FUNCTION Grey_To_Bin : INT // convert 4 bit grey code into 8 bit binary code
VAR_INPUT
	GreyBit0 : BOOL := FALSE ;
	GreyBit1 : BOOL := FALSE ;
	GreyBit2 : BOOL := FALSE ;
	GreyBit3 : BOOL := FALSE ;
END_VAR
VAR
	TempInt : INT ; // temporary 
END_VAR

// convert grey code into binary
TempInt.3 	:= GreyBit3 ;
TempInt.2	:= GreyBit3 	XOR GreyBit2 ;
TempInt.1	:= TempInt.2	XOR GreyBit1 ;
TempInt.0	:= TempInt.1	XOR GreyBit0 ;

Grey_To_Bin := TempInt ;

END_FUNCTION

(* stored: Version 1.1.0.1, ProductVersion 3.1.4024.3
   POU Grey_To_Bin: Id {b081e35e-5fed-49a3-83e6-052175f57bfb}, SpecialFunc None *)
